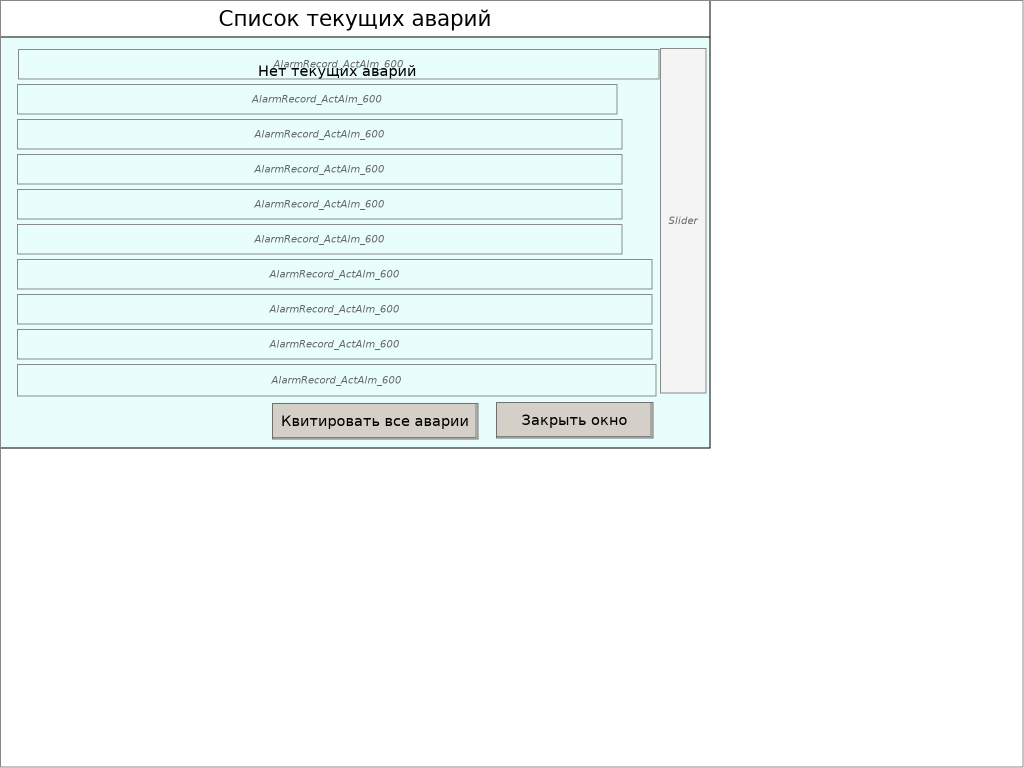
VISUALIZATION Current_Alarms_dialog  // 1024x768
    Rectangle (0,0 710x448)
    Frame (17,84 600x30)
        shows AlarmRecord_ActAlm_600(AlarmRecord := PRG_Alarms_Core.HMI_ActiveAlarms[2])
    Frame (17,119 605x30)
        shows AlarmRecord_ActAlm_600(AlarmRecord := PRG_Alarms_Core.HMI_ActiveAlarms[3])
    Frame (17,154 605x30)
        shows AlarmRecord_ActAlm_600(AlarmRecord := PRG_Alarms_Core.HMI_ActiveAlarms[4])
    Frame (17,189 605x30)
        shows AlarmRecord_ActAlm_600(AlarmRecord := PRG_Alarms_Core.HMI_ActiveAlarms[5])
    Frame (17,224 605x30)
        shows AlarmRecord_ActAlm_600(AlarmRecord := PRG_Alarms_Core.HMI_ActiveAlarms[6])
    Frame (17,259 635x30)
        shows AlarmRecord_ActAlm_600(AlarmRecord := PRG_Alarms_Core.HMI_ActiveAlarms[7])
    Frame (17,294 635x30)
        shows AlarmRecord_ActAlm_600(AlarmRecord := PRG_Alarms_Core.HMI_ActiveAlarms[8])
    Frame (17,329 635x30)
        shows AlarmRecord_ActAlm_600(AlarmRecord := PRG_Alarms_Core.HMI_ActiveAlarms[9])
    Frame (17,364 639x32)
        shows AlarmRecord_ActAlm_600(AlarmRecord := PRG_Alarms_Core.HMI_ActiveAlarms[10])
    Label (222,56 231x30), "Нет текущих аварий", invisible if: PRG_Alarms_Core.HMI_ActiveAlarms[1].isActive
    Frame (18,49 641x30)
        shows AlarmRecord_ActAlm_600(AlarmRecord := PRG_Alarms_Core.HMI_ActiveAlarms[1])
    Button (496,402 157x36), "Закрыть окно"
        OnMouseClick: CloseDialog Dialog=Current_Alarms_dialog, Result=OK, NumpadKeypadSet=True
    Button (272,403 206x36), "Квитировать все аварии"
        tap LibAlarm.bLocalQuitAllAlarms
    Rectangle (0,0 710x37), "Список текущих аварий"
    Slider (660,48 46x345), variable: PRG_Alarms_Core.HMI_CurShiftAA, scale 0..1000
END_VISUALIZATION

(* stored: Version 1.1.0.1, ProductVersion 3.1.4024.2
   Visu Current_Alarms_dialog: Id {06b1270d-1dd8-4f22-abb0-e26d5893b790} *)
